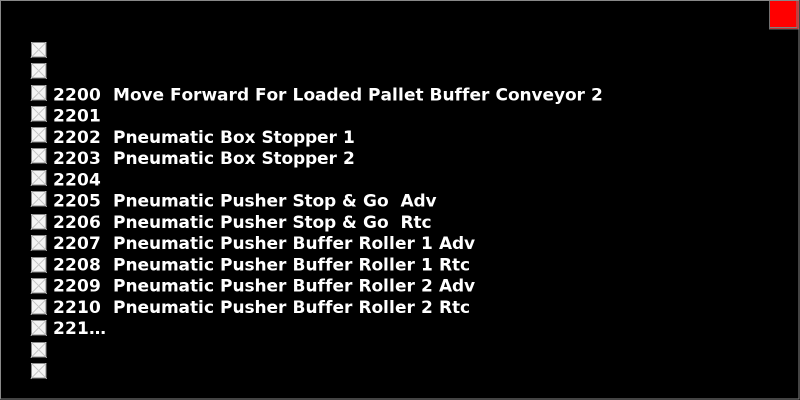
VISUALIZATION P2_DO3  // 800x400, background image 
    ImageSwitcher (31,42 15x15), variable: InputOutput_GVL.Digital_Output[33], behaviour: TOGGLE
    Label (50,16 625x391), "2200 Move Forward For Loaded Pallet Buffer Conveyor 2 2201 2202 Pneumatic Box Stopper 1 2203 Pneumatic Box Stopper 2 2204 2205 Pneumatic Pusher Stop & Go Adv 2206 Pneumatic Pusher Stop & Go Rtc 2207 Pneumatic Pusher Buffer Roller 1 Adv 2208 Pneumatic Pusher Buffer Roller 1 Rtc 2209 Pneumatic Pusher Buffer Roller 2 Adv 2210 Pneumatic Pusher Buffer Roller 2 Rtc 2211 2212 Interlock Status Infeed Modullar Busy 2213 Release Brake Motor Right Angle Lifter 2214 Interlock Request Pallet to Infeed Dispenser 2215 Interlock Request Pallet to Conveyor Outfeed Existing"
    ImageSwitcher (31,63 15x15), variable: InputOutput_GVL.Digital_Output[34], behaviour: TOGGLE
    ImageSwitcher (31,85 15x15), variable: InputOutput_GVL.Digital_Output[35], behaviour: TOGGLE
    ImageSwitcher (31,106 15x15), variable: InputOutput_GVL.Digital_Output[36], behaviour: TOGGLE
    ImageSwitcher (31,127 15x15), variable: InputOutput_GVL.Digital_Output[37], behaviour: TOGGLE
    ImageSwitcher (31,148 15x15), variable: InputOutput_GVL.Digital_Output[38], behaviour: TOGGLE
    ImageSwitcher (31,170 15x15), variable: InputOutput_GVL.Digital_Output[39], behaviour: TOGGLE
    ImageSwitcher (31,191 15x15), variable: InputOutput_GVL.Digital_Output[40], behaviour: TOGGLE
    ImageSwitcher (31,214 15x15), variable: InputOutput_GVL.Digital_Output[41], behaviour: TOGGLE
    ImageSwitcher (31,235 15x15), variable: InputOutput_GVL.Digital_Output[42], behaviour: TOGGLE
    ImageSwitcher (31,257 15x15), variable: InputOutput_GVL.Digital_Output[43], behaviour: TOGGLE
    ImageSwitcher (31,278 15x15), variable: InputOutput_GVL.Digital_Output[44], behaviour: TOGGLE
    ImageSwitcher (31,299 15x15), variable: InputOutput_GVL.Digital_Output[45], behaviour: TOGGLE
    ImageSwitcher (31,320 15x15), variable: InputOutput_GVL.Digital_Output[46], behaviour: TOGGLE
    ImageSwitcher (31,342 15x15), variable: InputOutput_GVL.Digital_Output[47], behaviour: TOGGLE
    ImageSwitcher (31,363 15x15), variable: InputOutput_GVL.Digital_Output[48], behaviour: TOGGLE
    Button (769,-1 30x30), image: VisuSymbols.Symbols.Wrong
        OnMouseClick: CloseDialog Dialog=P2_DO3, Result=OK, NumpadKeypadSet=True
END_VISUALIZATION

(* stored: Version 1.1.0.1, ProductVersion 3.1.4024.12
   Visu P2_DO3: Id {048e0ea5-2134-4cc5-a398-ec6f4dd8fc71} *)
